SYSTEM Example1
  (* Version 1.0, 2008-11-22, Goran Cengic, Chalmers *)
  DEVICE Test Device : DeviceType_not_used
    RESOURCE TestResource : ResourceType_not_used
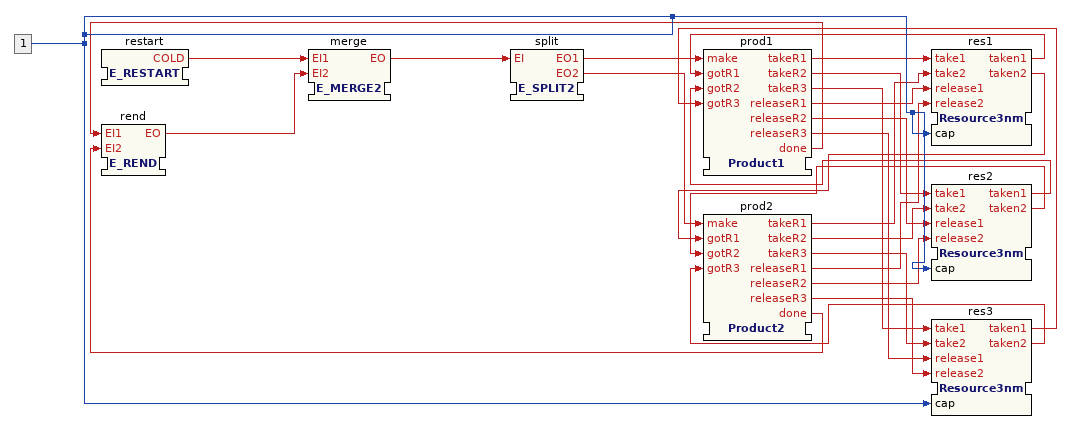
      FBS
        restart : E_RESTART;
        merge : E_MERGE2;
        split : E_SPLIT2;
        rend : E_REND;
        prod1 : Product1;
        prod2 : Product2;
        res1 : Resource3nm;
        res2 : Resource3nm;
        res3 : Resource3nm;
      END_FBS
      EVENT_CONNECTIONS
        restart.COLD TO merge.EI1;
        merge.EO TO split.EI;
        split.EO1 TO prod1.make;
        split.EO2 TO prod2.make;
        prod1.takeR1 TO res1.take1;
        prod1.takeR2 TO res2.take1;
        prod1.takeR3 TO res3.take1;
        prod1.releaseR1 TO res1.release1;
        prod1.releaseR2 TO res2.release1;
        prod1.releaseR3 TO res3.release1;
        res1.taken1 TO prod1.gotR1;
        res2.taken1 TO prod1.gotR2;
        res3.taken1 TO prod1.gotR3;
        prod2.takeR1 TO res1.take2;
        prod2.takeR2 TO res2.take2;
        prod2.takeR3 TO res3.take2;
        prod2.releaseR1 TO res1.release2;
        prod2.releaseR2 TO res2.release2;
        prod2.releaseR3 TO res3.release2;
        res1.taken2 TO prod2.gotR1;
        res2.taken2 TO prod2.gotR2;
        res3.taken2 TO prod2.gotR3;
        prod1.done TO rend.EI1;
        prod2.done TO rend.EI2;
        rend.EO TO merge.EI2;
      END_CONNECTIONS
      DATA_CONNECTIONS
        1 TO res1.cap;
        1 TO res2.cap;
        1 TO res3.cap;
      END_CONNECTIONS
    END_RESOURCE
  END_DEVICE
END_SYSTEM
(* other elements stored in the file *)
(* Product 1 *)
(* Product 2 *)
